ABB RobotStudio station: Robstu1.rsstnx

Station Project2 (saved by RobotStudio 25.3.11371.0)
Controller IRB660_180_315, task T_ROB1: task frame (RAPID world) sits at (0, 0, 0) mm, rotated rx 0 ry 0 rz 180 deg in the station
Controller IRB660_180_315
  mechanical unit ROB_1: IRB660_180_315__01, 6 joints, base frame (0, 0, 0) mm
Layout (positions relative to the parent item):
  - IRB660_180_315__01 [mechanism, from %ABB.RobotStudio.Models.IRB660%\IRB660_180_315__01.rslib] at (0, 0, 0) mm, rotated rx 0 ry 0 rz 180 deg; joint values [0, -0.3918, 0.0379, -0.0478] (rad or m)
  - CELDA_CON_BANDAS [part] at (-6782.38, -32.36, 0) mm, size 7936.5 x 10331 x 975 mm
  - Gripper [part] at (-1420.31, 0, 1684.89) mm, rotated rx -90 ry 0 rz 2.74 deg, size 289.7 x 128 x 268.8 mm
  - Carcasa [part] at (-1420.31, 0, 1684.89) mm, rotated rx 180 ry 0 rz 92.74 deg, size 250 x 250 x 150 mm
Attachment: Gripper is attached to IRB660_180_315__01 / Link6
Attachment: Carcasa is attached to Gripper
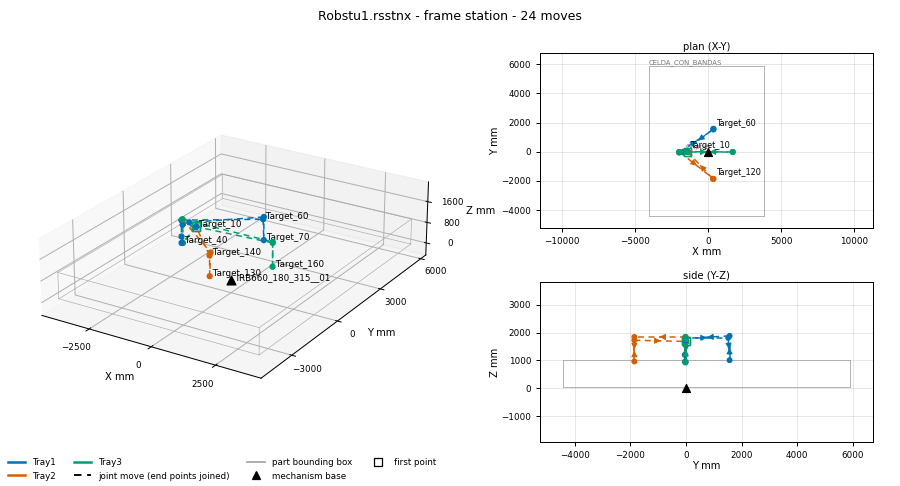
[picture p0: tool path of Robstu1.rsstnx in frame station, 24 of 24 moves have a stored position in this frame; points joined in program order, loops and branches not executed]
Targets, tools, work objects and paths stored in the station, written as RAPID:
! task T_ROB1
MODULE Module1
  CONST robtarget Target_10:=[[1420.311515248,0,1684.891137119],[0,-0.023885973,0.999714689,0],[0,0,-1,0],[9E+09,9E+09,9E+09,9E+09,9E+09,9E+09]];
  CONST robtarget Target_20:=[[1947.548961229,42.934299133,1656.651991798],[0,-0.02388597,0.99971469,0],[0,0,-1,0],[9E+09,9E+09,9E+09,9E+09,9E+09,9E+09]];
  CONST robtarget Target_30:=[[1998.576020327,42.934298907,1201.382064995],[0,-0.02388597,0.99971469,0],[0,0,-1,0],[9E+09,9E+09,9E+09,9E+09,9E+09,9E+09]];
  CONST robtarget Target_40:=[[1998.576031802,42.934299153,956.869146015],[0,-0.02388597,0.99971469,0],[0,0,-1,0],[9E+09,9E+09,9E+09,9E+09,9E+09,9E+09]];
  CONST robtarget Target_50:=[[1998.576023912,42.934298984,1815.390955495],[0,-0.02388597,0.99971469,0],[0,0,-1,0],[9E+09,9E+09,9E+09,9E+09,9E+09,9E+09]];
  CONST robtarget Target_60:=[[-356.834524529,-1518.833962005,1815.390949918],[0,-0.023885958,0.99971469,0],[-2,0,-2,0],[9E+09,9E+09,9E+09,9E+09,9E+09,9E+09]];
  CONST robtarget Target_70:=[[-356.834572385,-1568.833902067,1009.132998965],[0,-0.023885958,0.99971469,0],[-2,0,-2,0],[9E+09,9E+09,9E+09,9E+09,9E+09,9E+09]];
  CONST robtarget Target_80:=[[-356.834573872,-1568.833908603,1883.617999409],[0,-0.023885958,0.99971469,0],[-2,0,-2,0],[9E+09,9E+09,9E+09,9E+09,9E+09,9E+09]];
  CONST robtarget Target_90:=[[1687.428921426,17.397989448,1792.700063645],[0,-0.023885959,0.99971469,0],[0,0,-1,0],[9E+09,9E+09,9E+09,9E+09,9E+09,9E+09]];
  CONST robtarget Target_100:=[[1966.137023583,17.397990514,951.587909759],[0,-0.02388596,0.99971469,0],[0,0,-1,0],[9E+09,9E+09,9E+09,9E+09,9E+09,9E+09]];
  CONST robtarget Target_110:=[[1966.137028763,17.39799056,1845.778952192],[0,-0.02388596,0.99971469,0],[0,0,-1,0],[9E+09,9E+09,9E+09,9E+09,9E+09,9E+09]];
  CONST robtarget Target_120:=[[-368.07610741,1859.213917347,1845.778952941],[0,-0.023885958,0.99971469,0],[1,0,1,0],[9E+09,9E+09,9E+09,9E+09,9E+09,9E+09]];
  CONST robtarget Target_130:=[[-324.717035096,1859.2139052,963.347379517],[0,-0.023885958,0.99971469,0],[1,0,1,0],[9E+09,9E+09,9E+09,9E+09,9E+09,9E+09]];
  CONST robtarget Target_140:=[[-324.717036336,1859.213912297,1726.277956149],[0,-0.023885958,0.99971469,0],[1,0,1,0],[9E+09,9E+09,9E+09,9E+09,9E+09,9E+09]];
  CONST robtarget Target_150:=[[-1674.101919362,17.39806355,1845.778951015],[0,-0.023885958,0.99971469,0],[1,0,1,0],[9E+09,9E+09,9E+09,9E+09,9E+09,9E+09]];
  CONST robtarget Target_160:=[[-1674.101910758,17.398063461,924.890105022],[0,-0.023885958,0.99971469,0],[1,0,1,0],[9E+09,9E+09,9E+09,9E+09,9E+09,9E+09]];
  CONST robtarget Target_170:=[[-1674.101921351,17.398063571,1808.228026907],[0,-0.023885958,0.99971469,0],[1,0,1,0],[9E+09,9E+09,9E+09,9E+09,9E+09,9E+09]];
  PROC Tray1()
    MoveJ Target_10,v100,z100,tool0\WObj:=wobj0;
    MoveJ Target_20,v100,z100,tool0\WObj:=wobj0;
    MoveJ Target_30,v100,z100,tool0\WObj:=wobj0;
    MoveJ Target_40,v100,z100,tool0\WObj:=wobj0;
    MoveJ Target_50,v100,z100,tool0\WObj:=wobj0;
    MoveJ Target_60,v100,z100,tool0\WObj:=wobj0;
    MoveJ Target_70,v100,z100,tool0\WObj:=wobj0;
    MoveJ Target_80,v100,z100,tool0\WObj:=wobj0;
    MoveJ Target_90,v100,z100,tool0\WObj:=wobj0;
  ENDPROC
  PROC Tray2()
    MoveJ Target_10,v100,z100,tool0\WObj:=wobj0;
    MoveJ Target_100,v100,z100,tool0\WObj:=wobj0;
    MoveJ Target_110,v100,z100,tool0\WObj:=wobj0;
    MoveJ Target_120,v100,z100,tool0\WObj:=wobj0;
    MoveJ Target_130,v100,z100,tool0\WObj:=wobj0;
    MoveJ Target_140,v100,z100,tool0\WObj:=wobj0;
    MoveJ Target_10,v100,z100,tool0\WObj:=wobj0;
  ENDPROC
  PROC Tray3()
    MoveJ Target_10,v100,z100,tool0\WObj:=wobj0;
    MoveJ Target_10,v100,z100,tool0\WObj:=wobj0;
    MoveJ Target_100,v100,z100,tool0\WObj:=wobj0;
    MoveJ Target_110,v100,z100,tool0\WObj:=wobj0;
    MoveJ Target_150,v100,z100,tool0\WObj:=wobj0;
    MoveJ Target_160,v100,z100,tool0\WObj:=wobj0;
    MoveJ Target_170,v100,z100,tool0\WObj:=wobj0;
    MoveJ Target_10,v100,z100,tool0\WObj:=wobj0;
  ENDPROC
ENDMODULE

